Universal Robots PolyScope program: fun2.urp

Program fun2 (installation=default directory=/programs createdIn=5.9.1.1031110 lastSavedIn=5.9.1.1031110 robotSerialNumber=20195501059)
Calibrated DH parameters: a=[0.000146, -0.418764, -0.053981, 0.000058, -0.000023, 0]; d=[0.162545, 37.319448, -206.067439, 168.881546, 0.09955, 0.099464]; alpha=[1.57004, -0.001979, 0.002304, 1.570607, -1.57066, 0]; deltaTheta=[0, -0.174616, -1.258233, 1.432844, -0.000001, 0]
Robot Program (runOnlyOnce=true)
  URCap Gripper (Robotiq_Grippers, Robotiq Inc.) dataModel(position=100.0, force=100.0, speed=100.0, positionInDouble=100.0, forceInDouble=100.0, speedInDouble=100.0, slaveIds=[9], blocking=true)
  MoveL speed 250 mm/s, acceleration 1200 mm/s^2 (useActiveTCP=true) feature=Base
    Waypoint Waypoint_1: TCP in base x=107.129 y=-470.484 z=45.798 mm, rx=2.748 ry=1.5225 rz=0 rad; joints [86.738, -80.238, 122.137, -131.891, 270.057, -241.197] deg; TCP offset x=0 y=0 z=174 mm, rx=0 ry=0 rz=0 rad
  MoveL speed 250 mm/s, acceleration 1200 mm/s^2 (useActiveTCP=true) feature=Base
    Waypoint Waypoint_3: TCP in base x=271.683 y=-360.461 z=45.778 mm, rx=-2.748 ry=-1.5224 rz=-0.0001 rad; joints [109.776, -84.168, 126.847, -132.669, 270.07, -218.158] deg
  URCap Olis Teleop (Olis Teleop, Olis Robotics) dataModel(OperatorMessage=Teleoperation demo time!)
  MoveL speed 250 mm/s, acceleration 1200 mm/s^2 (useActiveTCP=true) feature=Base
    Waypoint Waypoint_1: TCP in base x=107.129 y=-470.484 z=45.798 mm, rx=2.748 ry=1.5225 rz=0 rad; joints [86.738, -80.238, 122.137, -131.891, 270.057, -241.197] deg
